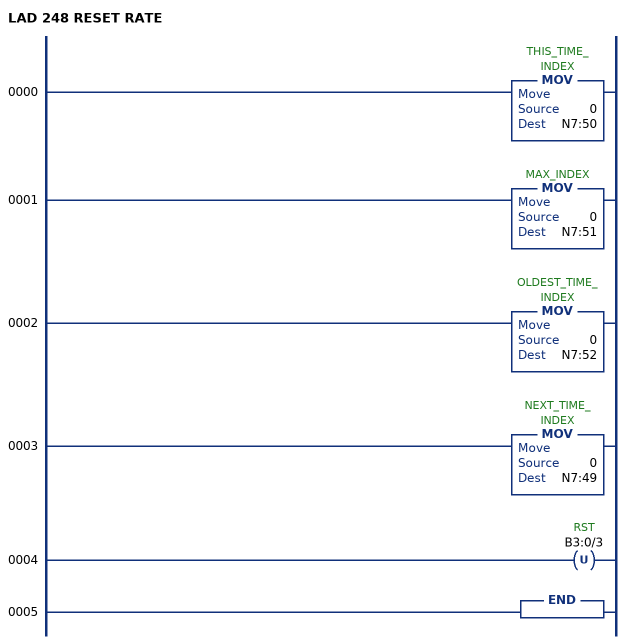
% Rung: 0 %
SOR MOV 0 N7:50 EOR
%   N7:50  THIS_TIME_INDEX %
% Rung: 1 %
SOR MOV 0 N7:51 EOR
%   N7:51  MAX_INDEX %
% Rung: 2 %
SOR MOV 0 N7:52 EOR
%   N7:52  OLDEST_TIME_INDEX %
% Rung: 3 %
SOR MOV 0 N7:49 EOR
%   N7:49  NEXT_TIME_INDEX %
% Rung: 4 %
SOR OTU B3:0/3 EOR
%   B3:0/3  RST %
% Rung: 5 %
SOR END EOR

LADDER 249 "NP STOP"    % stop on no good %
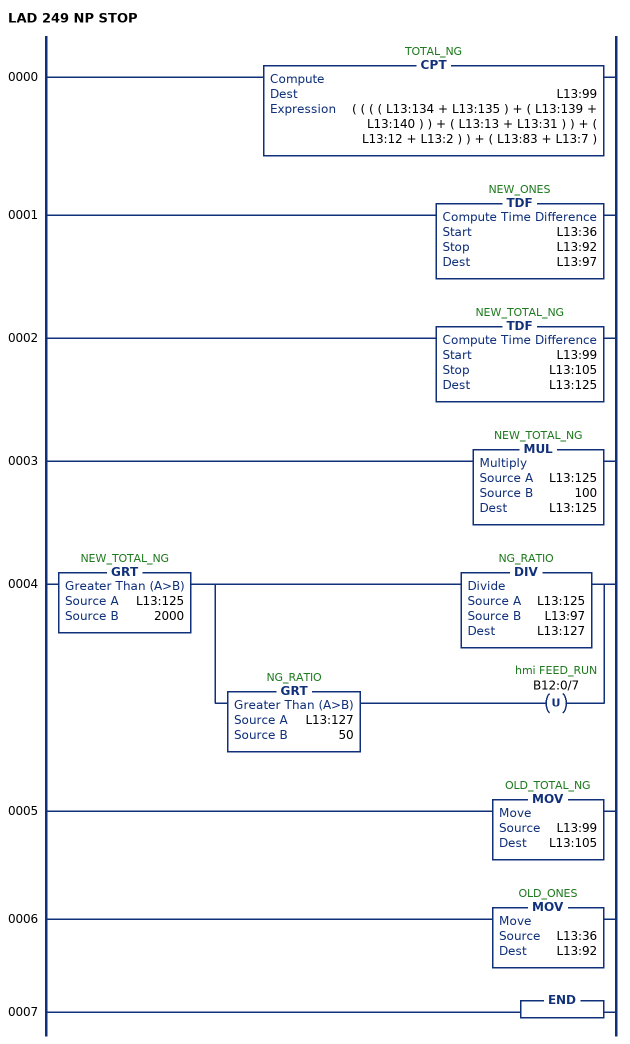
% Rung: 0 %
SOR CPT L13:99 " ( ( ( ( L13:134 + L13:135 ) + ( L13:139 + L13:140 ) ) + ( L13:13 + L13:31 ) ) + ( L13:12 + L13:2 ) ) + ( L13:83 + L13:7 ) " EOR
%   L13:99  TOTAL_NG %
%   L13:134  "too wide bottom" %
%   L13:135  "too close bottom" %
%   L13:139  "too close top count" %
%   L13:140  "too wide top count" %
%   L13:31  I5_SKIPPEDCOUNT %
%   L13:12  I6_SKIPPEDCOUNT %
%   L13:83  I5_FAIL_COUNT %
%   L13:7  I6_FAIL_COUNT %
% Rung: 1 %
SOR TDF L13:36 L13:92 L13:97 EOR
%   L13:36  ONES %
%   L13:92  OLD_ONES %
%   L13:97  NEW_ONES %
% Rung: 2 %
SOR TDF L13:99 L13:105 L13:125 EOR
%   L13:99  TOTAL_NG %
%   L13:105  OLD_TOTAL_NG %
%   L13:125  NEW_TOTAL_NG %
% Rung: 3 %
SOR MUL L13:125 100 L13:125 EOR
%   L13:125  NEW_TOTAL_NG %
% Rung: 4 %
SOR GRT L13:125 2000 BST DIV L13:125 L13:97 L13:127 NXB GRT L13:127 50 OTU B12:0/7 BND EOR
%   L13:125  NEW_TOTAL_NG %
%   L13:97  NEW_ONES %
%   L13:127  NG_RATIO %
%   B12:0/7  FEED_RUN  "hmi" %
% Rung: 5 %
SOR MOV L13:99 L13:105 EOR
%   L13:99  TOTAL_NG %
%   L13:105  OLD_TOTAL_NG %
% Rung: 6 %
SOR MOV L13:36 L13:92 EOR
%   L13:36  ONES %
%   L13:92  OLD_ONES %
% Rung: 7 %
SOR END EOR

LADDER 250 "SPEED BOT"    % high speed %
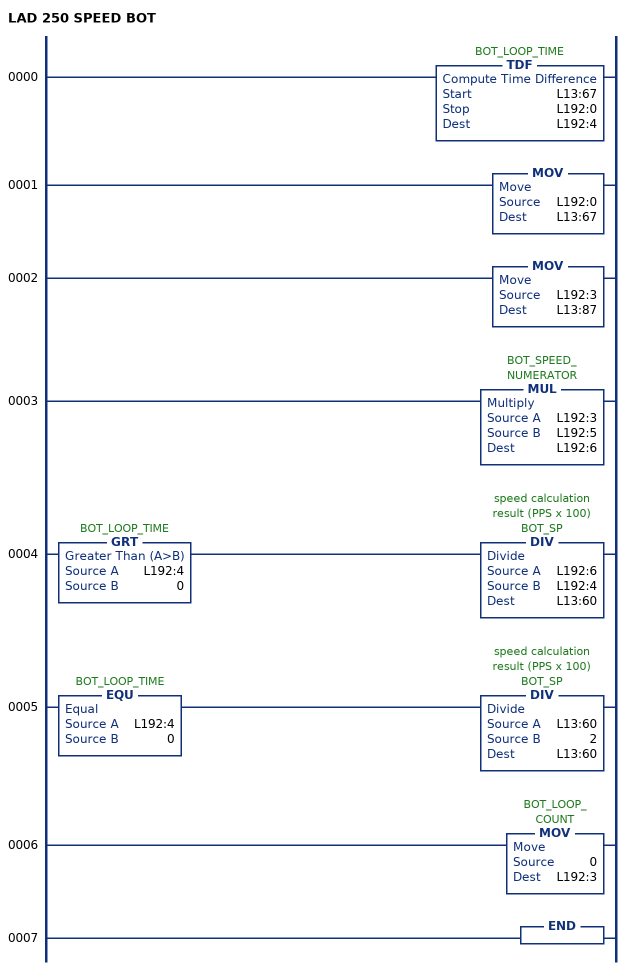
% Rung: 0 %
SOR TDF L13:67 L192:0 L192:4 EOR
%   L192:0  BOT_THIS_TIME  "rtc bot belt movement event time" %
%   L192:4  BOT_LOOP_TIME %
% Rung: 1 %
SOR MOV L192:0 L13:67 EOR
%   L192:0  BOT_THIS_TIME  "rtc bot belt movement event time" %
% Rung: 2 %
SOR MOV L192:3 L13:87 EOR
%   L192:3  BOT_LOOP_COUNT %
% Rung: 3 %
SOR MUL L192:3 L192:5 L192:6 EOR
%   L192:3  BOT_LOOP_COUNT %
%   L192:5  TKS_PER_SECOND %
%   L192:6  BOT_SPEED_NUMERATOR %
% Rung: 4 %
SOR GRT L192:4 0 DIV L192:6 L192:4 L13:60 EOR
%   L192:4  BOT_LOOP_TIME %
%   L192:6  BOT_SPEED_NUMERATOR %
%   L13:60  BOT_SP  "speed calculation result (PPS x 100)" %
% Rung: 5 %
SOR EQU L192:4 0 DIV L13:60 2 L13:60 EOR
%   L192:4  BOT_LOOP_TIME %
%   L13:60  BOT_SP  "speed calculation result (PPS x 100)" %
% Rung: 6 %
SOR MOV 0 L192:3 EOR
%   L192:3  BOT_LOOP_COUNT %
% Rung: 7 %
SOR END EOR

LADDER 251 "SPEED TOP"    % high speed %
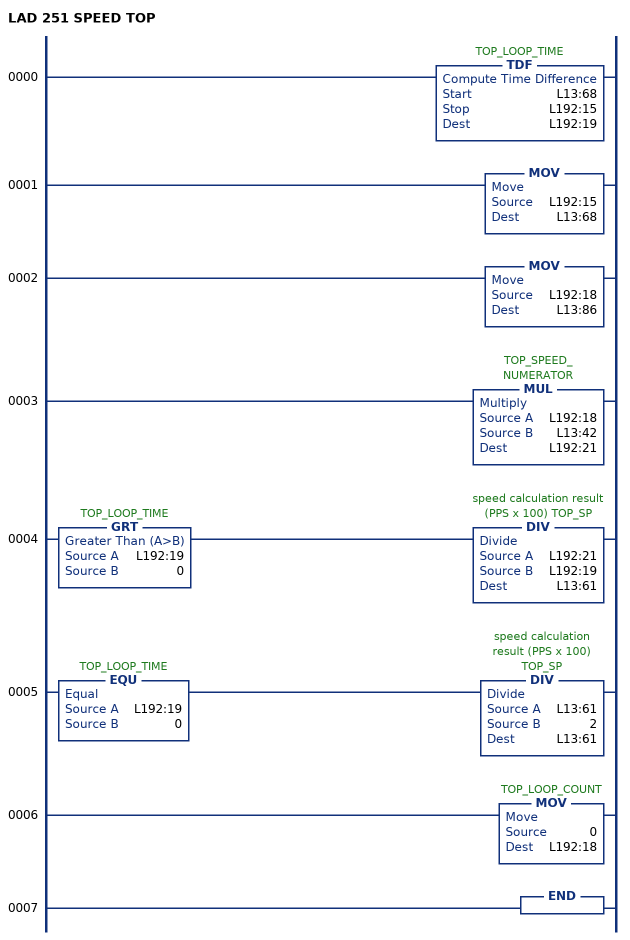
% Rung: 0 %
SOR TDF L13:68 L192:15 L192:19 EOR
%   L192:15  TOP_THIS_TIME  "rtc top belt movement event time" %
%   L192:19  TOP_LOOP_TIME %
% Rung: 1 %
SOR MOV L192:15 L13:68 EOR
%   L192:15  TOP_THIS_TIME  "rtc top belt movement event time" %
% Rung: 2 %
SOR MOV L192:18 L13:86 EOR
%   L192:18  TOP_LOOP_COUNT %
% Rung: 3 %
SOR MUL L192:18 L13:42 L192:21 EOR
%   L192:18  TOP_LOOP_COUNT %
%   L192:21  TOP_SPEED_NUMERATOR %
% Rung: 4 %
SOR GRT L192:19 0 DIV L192:21 L192:19 L13:61 EOR
%   L192:19  TOP_LOOP_TIME %
%   L192:21  TOP_SPEED_NUMERATOR %
%   L13:61  TOP_SP  "speed calculation result (PPS x 100)" %
% Rung: 5 %
SOR EQU L192:19 0 DIV L13:61 2 L13:61 EOR
%   L192:19  TOP_LOOP_TIME %
%   L13:61  TOP_SP  "speed calculation result (PPS x 100)" %
% Rung: 6 %
SOR MOV 0 L192:18 EOR
%   L192:18  TOP_LOOP_COUNT %
% Rung: 7 %
SOR END EOR

LADDER 252 "P BOT"    % high speed %
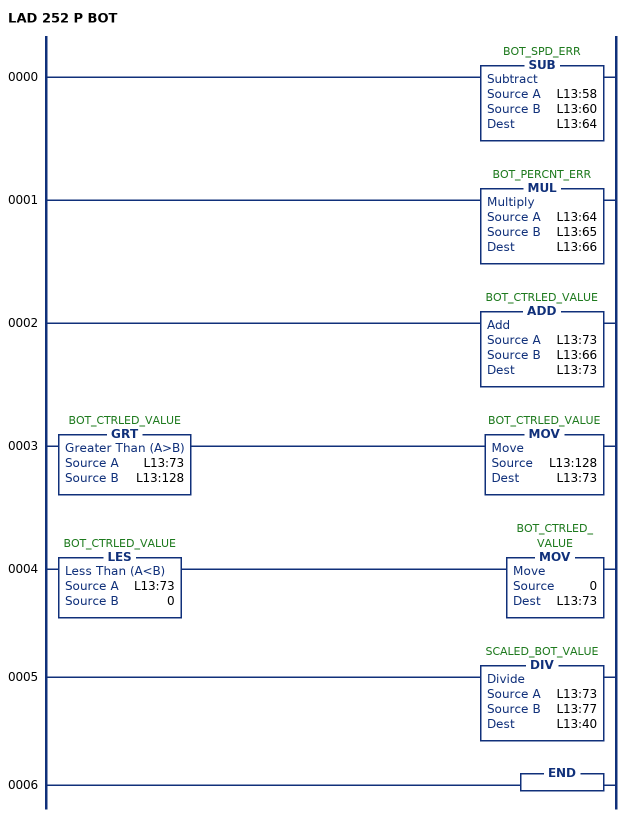
% Rung: 0 %
SOR SUB L13:58 L13:60 L13:64 EOR
%   L13:58  BOT_SPD_SETPOINT %
%   L13:60  BOT_SP  "speed calculation result (PPS x 100)" %
%   L13:64  BOT_SPD_ERR %
% Rung: 1 %
SOR MUL L13:64 L13:65 L13:66 EOR
%   L13:64  BOT_SPD_ERR %
%   L13:65  POS5SHIFT %
%   L13:66  BOT_PERCNT_ERR %
% Rung: 2 %
SOR ADD L13:73 L13:66 L13:73 EOR
%   L13:73  BOT_CTRLED_VALUE %
%   L13:66  BOT_PERCNT_ERR %
% Rung: 3 %
SOR GRT L13:73 L13:128 MOV L13:128 L13:73 EOR
%   L13:73  BOT_CTRLED_VALUE %
%   L13:128  "how much top has shifted since measurment" %
% Rung: 4 %
SOR LES L13:73 0 MOV 0 L13:73 EOR
%   L13:73  BOT_CTRLED_VALUE %
% Rung: 5 %
SOR DIV L13:73 L13:77 L13:40 EOR
%   L13:73  BOT_CTRLED_VALUE %
%   L13:40  SCALED_BOT_VALUE %
% Rung: 6 %
SOR END EOR

LADDER 253 "P TOP"    % high speed %
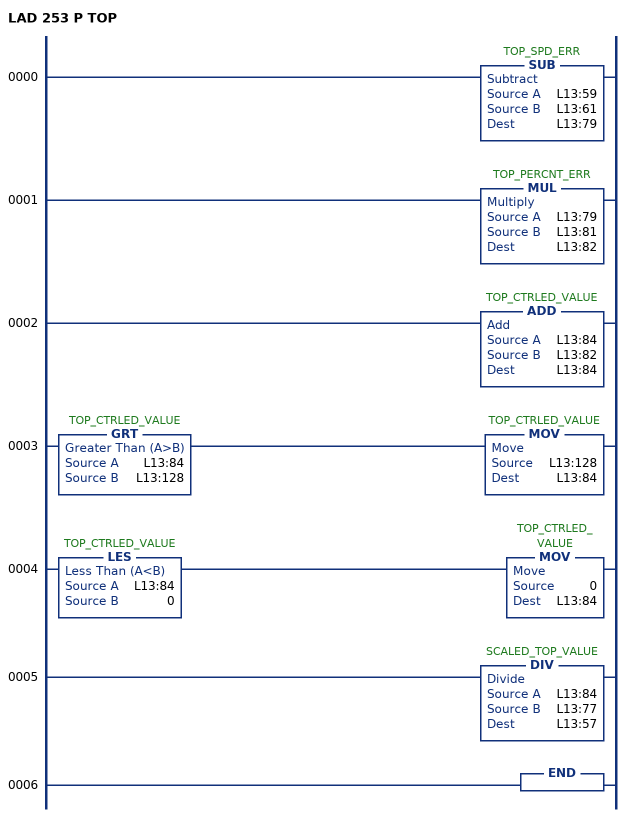
% Rung: 0 %
SOR SUB L13:59 L13:61 L13:79 EOR
%   L13:59  TOP_SPD_SETPOINT %
%   L13:61  TOP_SP  "speed calculation result (PPS x 100)" %
%   L13:79  TOP_SPD_ERR %
% Rung: 1 %
SOR MUL L13:79 L13:81 L13:82 EOR
%   L13:79  TOP_SPD_ERR %
%   L13:81  TOP_FDBK_RATIO %
%   L13:82  TOP_PERCNT_ERR %
% Rung: 2 %
SOR ADD L13:84 L13:82 L13:84 EOR
%   L13:84  TOP_CTRLED_VALUE %
%   L13:82  TOP_PERCNT_ERR %
% Rung: 3 %
SOR GRT L13:84 L13:128 MOV L13:128 L13:84 EOR
%   L13:84  TOP_CTRLED_VALUE %
%   L13:128  "how much top has shifted since measurment" %
% Rung: 4 %
SOR LES L13:84 0 MOV 0 L13:84 EOR
%   L13:84  TOP_CTRLED_VALUE %
% Rung: 5 %
SOR DIV L13:84 L13:77 L13:57 EOR
%   L13:84  TOP_CTRLED_VALUE %
%   L13:57  SCALED_TOP_VALUE %
% Rung: 6 %
SOR END EOR

LADDER 254 "TOTALCOUNT"
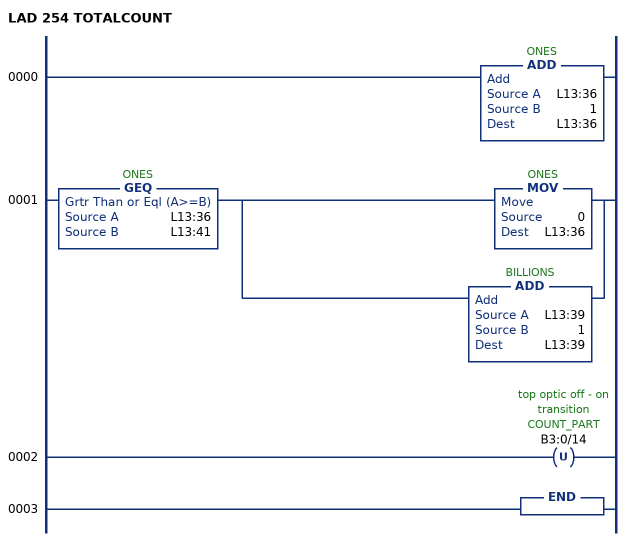
% Rung: 0 %
SOR ADD L13:36 1 L13:36 EOR
%   L13:36  ONES %
% Rung: 1 %
SOR GEQ L13:36 L13:41 BST MOV 0 L13:36 NXB ADD L13:39 1 L13:39 BND EOR
%   L13:36  ONES %
%   L13:41  "skipped count change in the last 3 seconds" %
%   L13:39  BILLIONS %
% Rung: 2 %
SOR OTU B3:0/14 EOR
%   B3:0/14  COUNT_PART  "top optic off - on transition" %
% Rung: 3 %
SOR END EOR

LADDER 255 "SAVED"
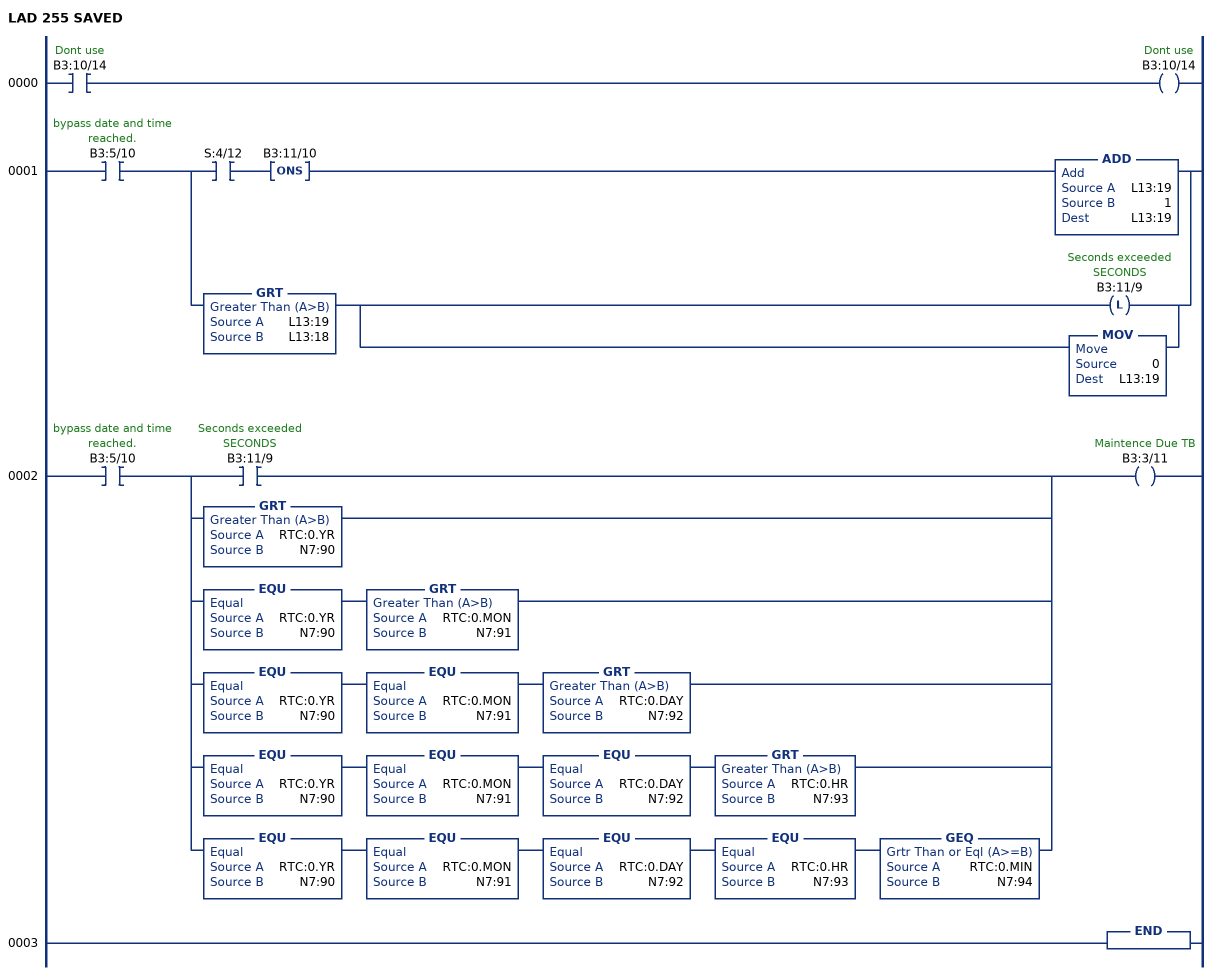
% Rung: 0 %
SOR XIC B3:10/14 OTE B3:10/14 EOR
%   B3:10/14  "Dont use" %
% Rung: 1 %
SOR XIC B3:5/10 BST XIC S:4/12 ONS B3:11/10 ADD L13:19 1 L13:19 NXB GRT L13:19 L13:18 BST OTL B3:11/9 NXB MOV 0 L13:19 BND BND EOR
%   B3:5/10  "bypass date and time reached." %
%   L13:18  MAX %
%   B3:11/9  SECONDS  "Seconds exceeded" %
% Rung: 2 %
SOR XIC B3:5/10 BST XIC B3:11/9 NXB GRT RTC:0.YR N7:90 NXB EQU RTC:0.YR N7:90 GRT RTC:0.MON N7:91 NXB EQU RTC:0.YR N7:90 EQU RTC:0.MON N7:91 GRT RTC:0.DAY N7:92 NXB EQU RTC:0.YR N7:90 EQU RTC:0.MON N7:91 EQU RTC:0.DAY N7:92 GRT RTC:0.HR N7:93 NXB EQU RTC:0.YR N7:90 EQU RTC:0.MON N7:91 EQU RTC:0.DAY N7:92 EQU RTC:0.HR N7:93 GEQ RTC:0.MIN N7:94 BND OTE B3:3/11 EOR
%   B3:5/10  "bypass date and time reached." %
%   B3:11/9  SECONDS  "Seconds exceeded" %
%   N7:90  RTC %
%   B3:3/11  TB  "Maintence Due" %
% Rung: 3 %
SOR END EOR

OTHER DOCUMENTED ADDRESSES
  B189:0/0  "change box"
  B189:0/9  "override boxing ok or not full signal"
  B189:0/11  "HMI force door close"
  B196:1/0  "Chute door is closed"
  B196:1/1  "control chute door"
  B196:1/13  "force box conveyor on"
  B196:3/0  "for hmi to continue production unlatched by hmi"
  HSC:0.0  "top"
  HSC:0.3/6  "Underflow interrupt"
  HSC:0.3/7  "Overflow interrupt"
  HSC:1.0  "bot"
  HSC:1.3/6  "Underflow interrupt"
  HSC:1.3/7  "Overflow interrupt"
  I:0.0/0  TOP_ENC
  I:0.0/2  CHUTE_OPTIC
  I:0.0/4  BOT_ENC
  I:0.0/10  PART_LONG
  I:0.0/12  INS_3_7_ACQ
  I:0.1/0  BOT_TRIG_OPTIC  "we don't need a bottom trigger!"
  I:0.1/1  INS_3_7_GOOD
  I:0.1/2  INS_3_7_NG
  I:0.1/4  "not used"
  I:0.1/5  "not used"
  I:0.1/6  "not used"
  I:0.1/7  "not used"
  I:0.1/8  "not used"
  I:0.1/9  "not used"
  I:0.1/10  "not used"
  I:0.1/11  "not used"
  I:0.1/12  "not used"
  I:0.1/13  "not used"
  I:0.1/14  "not used"
  I:0.1/15  "not used"
  I:0.2  "not used"
  I:0.2/3  "Packaging Conveyor full"
  I:0.2/4  "Packaging Conveyor Box in Position"
  I:0.3  "not used"
  I:0.4  "Spare Analog Input 1"
  I:0.5  "Spare Analog Input 2"
  I:0.6  "Spare Analog Input 3"
  I:2.0/0  FRONT_ESTOP
  I:2.0/1  REAR_ESTOP
  I:2.0/2  PACKAGER_CONNECTED
  I:2.0/3  BOX_CNV_NOT_FULL  "input turns off when box discharge full optics are blocked"
  I:2.0/4  BOX_NOT_IN_POS  "this input is on when a box is not in position"
  I:2.0/5  MCR
  I:2.0/6  MPCE  "primary safety relay on(e-stop)"
  I:2.0/7  MSCE  "secondary safety relay on(door) ce models only"
  I:2.0/8  FRONT_DOOR  "front door signal ce models only"
  I:2.0/9  REAR_DOOR  "rear door signal ce models only"
  I:2.0/10  MAINTENANCE_KEY_SW  "Maintenance Key Switch ce models only"
  I:2.0/11  "spare"
  I:2.0/12  "spare"
  I:2.0/13  FDER_PDL_SW  "Feeder Bowl Paddle Switch"
  I:2.0/14  "spare"
  I:2.0/15  TRACK_SENSOR  "Feeder Bowl Downtrack Sensor"
  L13:180  "maximum time between triggers"
  L13:181  "minimum okay time between triggers"
  L13:182  RATE_QUEUE_LIMIT
  L13:184  "intermediate i1 trig avg"
  L13:185  I1_TBT  "i1 average time between triggers"
  L13:186  "intermediate i5 trig avg"
  L13:187  I5_TBT  "i5 average time between triggers"
  L13:188  "intermediate i6 trig avg"
  L13:189  I6_TBT  "i6 average time between triggers"
  L13:190  "i1 timed q limit"
  L13:191  "i1 absolute q limit"
  L16:2  TRIG_DELAY_Q_MULTI
  L16:3  TRIG_DELAY_MIN_TIME
  L16:4  TRIG_DELAY_FLAT_RATE
  L16:5  CLEARTIME1  "time to clear tracking data"
  L16:6  CLEARTIME5
  L16:7  CLEARTIME6
  L16:8  PASS1PRTLOC
  L16:9  PASS1PROCESSTM
  L16:11  PASS5PROCESSTM
  L16:13  PASS6PROCESSTM
  L23:19  TOP_OPT_FAIL_CT
  L23:34  AIR_PRESSURE_FAULT
  L28:0  INS_1_TIME
  L29:0  INS_1_POS
  L30:0  INS_5_TIME
  L31:0  INS_5_POS
  L32:0  INS_6_TIME
  L33:0  INS_6_POS
  L192:1  BOT_LAST_TIME  "rtc bot belt previous movement event time"
  L192:2  BOT_CYCLE_TIME  "rtc bot belt time between events"
  L192:7  FROM_REAL  "distance from real part signal at optic location"
  L192:8  FROM_TRACKED  "distance from tracked part signal at optic location"
  L192:16  TOP_LAST_TIME  "rtc top belt previous movement event time"
  L192:17  TOP_CYCLE_TIME  "rtc top belt time between events"
  L199:5  ACQTM51
  L199:6  ACQTM52
  L199:7  ACQTM53
  L199:9  "ones"
  L199:10  "billions"
  L199:13  DUMP_LONG
  L199:15  ACQTM11
  L199:16  ACQTM12
  L199:17  ACQTM13
  L199:20  RESULTTM1
  L199:22  CLEARTIME5COUNT
  L199:23  CLEARTIME6COUNT
  L199:24  ACQTM61
  L199:25  ACQTM62
  L199:26  ACQTM63
  L199:27  TMSINCETRIG1
  L199:29  TMSINCETRIG5
  L199:30  TMSINCETRIG6
  L199:31  CLEARTIME1COUNT
  L199:32  RESULTTM5
  L199:33  RESULTTM6
  L199:34  MAXACQTM1
  L199:36  MAXACQTM6
  N15:5  INS_1_TRIG_LOC
  O:0.0/0  BELTS_ENABLE
  O:0.0/1  "spare"
  O:0.0/11  "Spare"
  O:0.0/12  "not used"
  O:0.0/13  "not used"
  O:0.0/14  "not used"
  O:0.0/15  "not used"
  O:0.1  "not used"
  O:0.2  "not used"
  O:0.3  "not used"
  PFILE:6  "check for part jams"
  PFILE:10  "Bottom belt HSC"
  PFILE:12  "Top belt HSC"
  Q2:55  END_OF_MAIN
  Q5:94  END_OF_BELTS
  T20:0  "Trigger On Time"
  U:9  "slow data"
  U:24  "check skipped fail rate"
  U:28  "faults"
  U:29  "speed"
  U:30  "count"
  U:31  "rate calc"
  U:32  "boxer"
  U:33  "bulk pack"
  U:34  "customer boxing unit signals"
  U:35  "cleanup"

REVISION NOTES
  13: updated count reset
  14: added io moduals
  15: multiple steps toward new hmi integration
  21: test
  27: fix error if bulk pack and no boxing fallout were on

DATA TABLE (non-zero values as saved)
DATA B3
% B3:0 % 0X80A0 0X0260 0X4080 0XA409 0X0EE5 0X1550 0X0804 0X0421 0X4F80 0X2550
% B3:10 % 0X2000 0X0006 0X1000 0X0000
DATA T4
% .PRE .ACC %
% T4:0 % 0 2
% T4:1 % 150 0
% T4:2 % 400 0
% T4:3 % 222 0
% T4:4 % 300 0
% T4:5 % 5 5
% T4:6 % 10 32766
% T4:7 % 666 0
% T4:8 % 20 14
% T4:9 % 50 9
% T4:10 % 200 0
% T4:11 % 111 0
% T4:12 % 55 267
% T4:13 % 250 0
% T4:14 % 666 0
% T4:15 % 1000 1635
% T4:16 % 400 0
% T4:17 % 100 41
% T4:18 % 5 0
% T4:19 % 300 0
% T4:20 % 200 0
% T4:21 % 200 0
% T4:22 % 200 0
% T4:23 % 250 0
% T4:24 % 666 0
% T4:25 % 666 0
% T4:26 % 666 0
% T4:27 % 250 0
% T4:28 % 250 0
% T4:29 % 5000 0
% T4:30 % 222 0
% T4:31 % 222 0
% T4:32 % 222 0
% T4:33 % 222 0
DATA C5
% .PRE .ACC %
% C5:0 % 32766 0
DATA R6
% .LEN .POS %
% R6:0 % 1250 0
% R6:1 % 1250 0
% R6:2 % 1024 0
% R6:3 % 1024 0
% R6:4 % 1250 0
% R6:5 % 1250 0
% R6:6 % 1713 0
% R6:7 % 1024 0
% R6:8 % 1024 0
% R6:9 % 3 0
% R6:10 % 1713 0
% R6:11 % 1713 0
% R6:12 % 10 0
% R6:13 % 10 0
% R6:14 % 10 0
% R6:15 % 10 0
% R6:16 % 1713 0
% R6:17 % 1713 0
% R6:18 % 1713 0
% R6:19 % 10 0
DATA N7
% N7:0 % 181 3 306 300 18 400 0 32767 500 500
% N7:10 % 1000 18 0 2 46 20 1000 2000 50 1050
% N7:20 % 32767 222 10 222 222 46 48 0 48 250
% N7:30 % 666 506 150 0 0 551 34 1 0 1
% N7:40 % 3 44 2 42 421 482 560 632 1636 0
% N7:50 % 0 0 0 16 1 1024 0 0 32766 18
% N7:60 % 1713 1713 1713 1021 1034 1024 4999 5 400 400
% N7:70 % 100 200 300 400 90 190 290 390 223 1082
% N7:80 % 0 0 32767 780 832 844 45 25 0 0
% N7:90 % 2011 4 4 12 1 45 25 222 222 12
% N7:100 % 1003 90 110 100 175 25 0 0 0 0
DATA F8
% F8:0 % 6 1 23807 499 0.23807
% F8:5 % 0 0 500 1.9 2
% F8:10 % 1 0.08897486 3058 101 63.26563
% F8:15 % 37.73437 4040 2 0 0
% F8:20 % 0 0.02 0 1 0
% F8:25 % 0 932781 0.222 279.6551 848597
% F8:30 % 0 170 0.03 38 852060
% F8:35 % 0 0 0 0 77
% F8:40 % 101 37.73437 0 100 1
% F8:45 % 1 2 0.21455 0 0
% F8:50 % 0 0 1 0 1
% F8:55 % 2000000 -221 0 0 0
% F8:95 % 0 0 0 492 4.92
DATA B12
% B12:0 % 0X6004 0X0000 0X0000 0X0000 0X0000 0X0000 0X0000 0X0000 0X0000 0X0000
DATA L13
% L13:0 % 14459 15864 0 23287 30394
% L13:5 % 10529 15570 0 26000 22358
% L13:10 % 23035 283076525 2480 15 90
% L13:15 % 1096044215 -2147483648 2147483647 2147483647 82058
% L13:20 % 1326931947 1686418909 777 1326019296 100
% L13:25 % 153441500 49 684 0 409304644
% L13:30 % 686738858 762 60000 409312962 444
% L13:35 % 6 88734 0 0 0
% L13:40 % 0 1000000000 1000000 409312904 409313893
% L13:45 % 409313944 150 0 58 1612026828
% L13:50 % 686729499 686730677 410822522 371 0
% L13:55 % 686728333 6 3782 0 500
% L13:60 % 0 1 58 600 0
% L13:65 % 100 0 2044072 79142050 -942969229
% L13:70 % 1612034666 24 32 0 1612026828
% L13:75 % 32 60 100 410822233 -6
% L13:80 % 24 74 -444 7 378216
% L13:85 % 74392164 0 0 0 5
% L13:90 % 10 5 88734 10 409313918
% L13:95 % 685935457 573 0 409313968 3334
% L13:100 % 3200 6 3100 14 227
% L13:105 % 3334 31 1326019172 133426 1326019166
% L13:110 % 6 100 50 1328950220 1612026733
% L13:115 % 1612026745 12 6 1612026739 2
% L13:120 % 0 202 50 100 47
% L13:125 % 0 1612034666 -7200 3276500 357468689
% L13:130 % 2 2 0 99 0
% L13:135 % 0 0 74392164 5 70
% L13:140 % 0 5 36 50 50
% L13:145 % 5 5 5 5 74373084
% L13:150 % 12 20 133420 -133420 283076525
% L13:155 % 0 -9 0 0 4589052
% L13:160 % 24 25 24 25 24
% L13:165 % 1612027177 1612027195 1612027177 1612027195 1026
% L13:170 % 6182 571 571 2147483647 4700
% L13:175 % 3760917 8 42 23 38
% L13:180 % 176247033 25 99000 52866 644409
% L13:185 % 64 916459 92 627156 63
% L13:190 % 4 5 0 0 0
DATA F14
% F14:0 % 1.32889e-38 5747.126 1550 1550 1638.3
% F14:5 % 1638.3 1638.3 1638.3 0 0
DATA N15
% N15:0 % 738 756 963 560 389 105 66 1199 300 10
% N15:10 % 71 887 0 0 0 0 1356 0 0 0
DATA L16
% L16:0 % 16 55 11 0 20
% L16:5 % 250 5000 5000 182 19
% L16:10 % 1256 18 2045 6599584 98
% L16:15 % 99 0 0 0 0
DATA L19
% L19:0 % 409304644 409305367 409305722 409305964 409306670
% L19:5 % 409307037 409307371 409307825 409308402 409309463
% L19:10 % 409310059 409310531 409311029 409311341 409311683
% L19:15 % 409312096 409312671 0 0 0
DATA L20
% L20:0 % 409296629 409296845 409297075 409297298 409297514
% L20:5 % 409297750 409298004 409298285 409298546 409299059
% L20:10 % 409299475 409299997 409300464 409301025 409301246
% L20:15 % 409301618 409301838 409302071 409302397 409302632
% L20:20 % 409302865 409303137 409303562 409303854 409304199
% L20:25 % 409304447 409304882 409305158 409305588 409305870
% L20:30 % 409306592 409306945 409307187 409307893 409308261
% L20:35 % 409308592 409309049 409309628 409310687 409311283
% L20:40 % 409311753 409312251 409312564 409312906 409313322
% L20:45 % 409313893 409295719 409295940 409296162 409296383
DATA L21
% L21:0 % 1612021086 1612021162 1612021243 1612021322 1612021398
% L21:5 % 1612021481 1612021571 1612021670 1612021762 1612021943
% L21:10 % 1612022090 1612022274 1612022439 1612022637 1612022715
% L21:15 % 1612022846 1612022924 1612023006 1612023121 1612023204
% L21:20 % 1612023286 1612023382 1612023532 1612023635 1612023757
% L21:25 % 1612023844 1612023998 1612024095 1612024247 1612024346
% L21:30 % 1612024601 1612024726 1612024811 1612025060 1612025190
% L21:35 % 1612025307 1612025468 1612025672 1612026046 1612026256
% L21:40 % 1612026422 1612026598 1612026708 1612026829 1612026975
% L21:45 % 1612027177 1612020765 1612020843 1612020921 1612020999
DATA L22
% L22:0 % 409302916 409303188 409303614 409303904 409304251
% L22:5 % 409304498 409304934 409305209 409305639 409305921
% L22:10 % 409306643 409306996 409307238 409307944 409308312
% L22:15 % 409308643 409309100 409309679 409310738 409311333
% L22:20 % 409311805 409312303 409312615 409312957 409313373
% L22:25 % 409313944 409295770 409295991 409296213 409296433
% L22:30 % 409296680 409296896 409297126 409297349 409297565
% L22:35 % 409297801 409298055 409298336 409298596 409299110
% L22:40 % 409299526 409300048 409300516 409301076 409301297
% L22:45 % 409301669 409301889 409302123 409302448 409302683
DATA L23
% L23:0 % 1612023304 1612023400 1612023550 1612023653 1612023775
% L23:5 % 1612023862 1612024016 1612024113 1612024265 1612024364
% L23:10 % 1612024619 1612024744 1612024829 1612025078 1612025208
% L23:15 % 1612025325 1612025486 1612025690 1612026064 1612026274
% L23:20 % 1612026440 1612026616 1612026726 1612026847 1612026993
% L23:25 % 1612027195 1612020783 1612020861 1612020939 1612021017
% L23:30 % 1612021104 1612021180 1612021261 1612021340 1612021416
% L23:35 % 1612021499 1612021589 1612021688 1612021780 1612021961
% L23:40 % 1612022108 1612022292 1612022457 1612022655 1612022733
% L23:45 % 1612022864 1612022942 1612023024 1612023139 1612023222
DATA L30
% L30:0 % 409312331 409312904 409294731 409294951 409295172
% L30:5 % 409295394 409295640 409295855 409296086 409296310
% L30:10 % 409296524 409296760 409297015 409297295 409297557
% L30:15 % 409298069 409298487 409299008 409299475 409300037
% L30:20 % 409300257 409300629 409300849 409301081 409301408
% L30:25 % 409301643 409301875 409302148 409302572 409302865
% L30:30 % 409303210 409303457 409303893 409304168 409304599
% L30:35 % 409304879 409305602 409305957 409306197 409306903
% L30:40 % 409307272 409307604 409308060 409308637 409309699
% L30:45 % 409310294 409310763 409311263 409311574 409311918
DATA L31
% L31:0 % 1612026626 1612026828 1612020416 1612020494 1612020572
% L31:5 % 1612020650 1612020737 1612020813 1612020894 1612020973
% L31:10 % 1612021049 1612021132 1612021222 1612021321 1612021413
% L31:15 % 1612021594 1612021741 1612021925 1612022090 1612022288
% L31:20 % 1612022366 1612022497 1612022575 1612022657 1612022772
% L31:25 % 1612022855 1612022937 1612023033 1612023183 1612023286
% L31:30 % 1612023408 1612023495 1612023649 1612023746 1612023898
% L31:35 % 1612023997 1612024252 1612024377 1612024462 1612024711
% L31:40 % 1612024841 1612024958 1612025119 1612025323 1612025697
% L31:45 % 1612025907 1612026073 1612026249 1612026359 1612026480
DATA L32
% L32:0 % 410812905 410813134 410813360 410813586 410813812
% L32:5 % 410814040 410814267 410814494 410814722 410814949
% L32:10 % 410815175 410815403 410815629 410815857 410816084
% L32:15 % 410816311 410816539 410816767 410816994 410817223
% L32:20 % 410817450 410817678 410817903 410818131 410818358
% L32:25 % 410818585 410818812 410819038 410819264 410819490
% L32:30 % 410819716 410819943 410820170 410820396 410820624
% L32:35 % 410820850 410821076 410821304 410821530 410821756
% L32:40 % 410821982 410822209 410822522 410822660 410822887
% L32:45 % 410811773 410811998 410812225 410812453 410812679
DATA L33
% L33:0 % 1612034666 1612034666 1612034666 1612034666 1612034666
% L33:5 % 1612034666 1612034666 1612034666 1612034666 1612034666
% L33:10 % 1612034666 1612034666 1612034666 1612034666 1612034666
% L33:15 % 1612034666 1612034666 1612034666 1612034666 1612034666
% L33:20 % 1612034666 1612034666 1612034666 1612034666 1612034666
% L33:25 % 1612034666 1612034666 1612034666 1612034666 1612034666
% L33:30 % 1612034666 1612034666 1612034666 1612034666 1612034666
% L33:35 % 1612034666 1612034666 1612034666 1612034666 1612034666
% L33:40 % 1612034666 1612034666 1612034666 1612034666 1612034666
% L33:45 % 1612034666 1612034666 1612034666 1612034666 1612034666
DATA B38
% B38:10 % 0X0000 0X0000 0X0000 0X0000 0X0000 0X0000 0X0000 0X0000 0XE000 0XFFFE
% B38:20 % 0X007C 0X2000 0X0000 0X0000 0X0000 0X0000 0X0000 0X0000 0X0000 0X0000
% B38:60 % 0X0000 0X0000 0X0000 0X8800 0X0003 0X0000 0X0FFF 0X0000 0X0000 0X0000
% B38:120 % 0X0000 0X0000 0X0000 0X0000 0X0000 0X0000 0X0000 0X0002
DATA B40
% B40:10 % 0X0000 0X0000 0X0000 0X0000 0X0000 0X0000 0X0000 0X0000 0XE000 0XFFFE
% B40:20 % 0X007C 0X2000 0X0000 0X0000 0X0000 0X0000 0X0000 0X0000 0X0000 0X0000
% B40:60 % 0X0000 0X0000 0X0000 0X8800 0X0003 0X0000 0X0FFF 0X0000 0X0000 0X0000
% B40:120 % 0X0000 0X0000 0X0000 0X0000 0X0000 0X0000 0X0000 0X0002
DATA L192
% L192:0 % 2044072 266932201 5055 0 0
% L192:5 % 1000000 0 999 999 8
% L192:10 % 0 0 0 78 17
% L192:15 % 79142050 332250347 860888 0 0
% L192:20 % 180 0 0 0 0
DATA B196
% B196:0 % 0X0814 0X9FFE 0X0005 0X0000 0X0000 0X0000 0X0000 0X0000 0X0000 0X0000
% B196:30 % 0XE800 0X9BFF 0XEBFF 0XFFDF 0XFFFF 0X0000 0X0000 0X0000 0X0000 0X0000
DATA L199
% L199:0 % 1 0 0 0 0
